// Mitsubishi GX Works2 project: ServMotor3   PLC: Q03UDV

PROGRAM MAIN
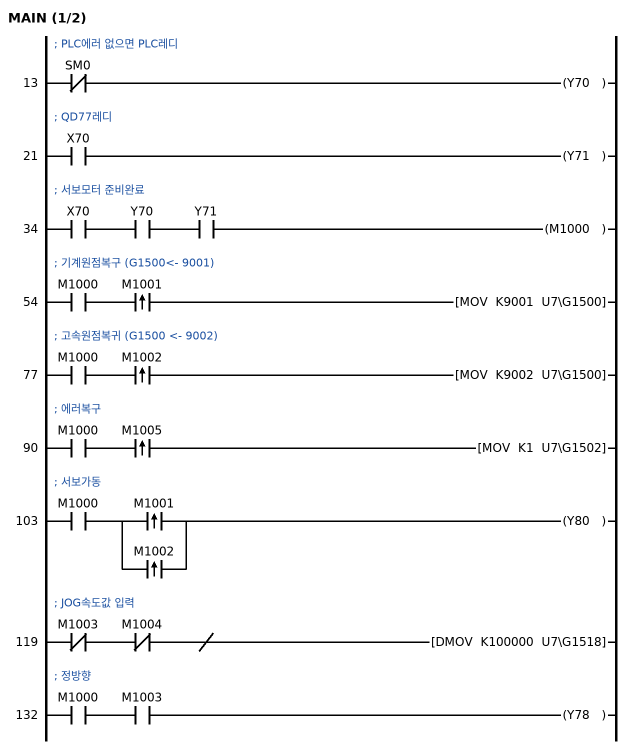
; PLC에러 없으면 PLC레디
13    LDI     SM0
      OUT     Y70
; QD77레디
21    LD      X70
      OUT     Y71
; 서보모터 준비완료
34    LD      X70
      AND     Y70
      AND     Y71
      OUT     M1000
; 기계원점복구 (G1500<- 9001)
54    LD      M1000
      ANDP    M1001
      MOV     K9001 U7\G1500
; 고속원점복귀 (G1500 <- 9002)
77    LD      M1000
      ANDP    M1002
      MOV     K9002 U7\G1500
; 에러복구
90    LD      M1000
      ANDP    M1005
      MOV     K1 U7\G1502
; 서보가동
103   LD      M1000
      LDP     M1001
      ORP     M1002
      ANB
      OUT     Y80
; JOG속도값 입력
119   LDI     M1003
      ANI     M1004
      INV
      DMOV    K100000 U7\G1518
; 정방향
132   LD      M1000
      AND     M1003
      OUT     Y78
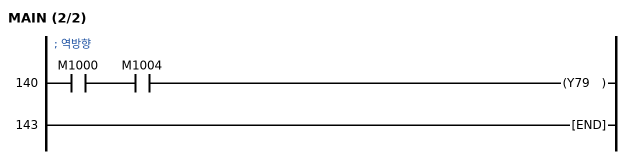
; 역방향
140   LD      M1000
      AND     M1004
      OUT     Y79
143   END
END_PROGRAM
